TYPE (* A Structure with 1 Bit *)
  (* Version 1.0, 2024-02-21, franz *)
  ST01B : STRUCT
    B_00 : BOOL; (* BIT 00 *)
  END_STRUCT;
END_TYPE
